(* IEC 61131-3 sources: CodesysTest/alpha/export/Device.dev/Plc Logic/Application/FBs/Motors/Applied Motion/FB_AppliedMotionBagDeliveryMotor_1.pou, 1 file *)

(* ---- SetRearMotorToTorqueMode.m.st ---- *)
(*#-#-#-#-#-#-#-#-#-#---Declaration---#-#-#-#-#-#-#-#-#-#-#-#-#*)

METHOD SetRearMotorToTorqueMode
VAR_INPUT
END_VAR
(*#-#-#-#-#-#-#-#-#-#---Implementation---#-#-#-#-#-#-#-#-#-#-#-#-#*)

sclCommand := 16#534F; // Output on
parameter1 := 16#4CB2;

commandSuccessful := FALSE;
commands.SendHostCommand := TRUE;
